PROGRAM Stn053_19_GrnRedRecircMergeSpurPrestop
VAR

	{attribute 'TcLinkToOSO' := '.iPuckPresent := <0,1,0>TIIB[N46S00 (AL1332)]^N46S03 (AL2341)^TxPDO^input byte 0;
								 .iBufferFull := <0,1,2>TIIB[N32S00 (AL1332)]^N32S05 (AL2341)^TxPDO^input byte 2;
								 .oStopLower := <0,1,4>TIIB[N46S00 (AL1332)]^N46S02 (EX260)^RxPDO^output byte 0'}
	fbConvStop: FB_ConvStop;
END_VAR

//MergeGrntoRedMergeSpurPrestopGrn  (3A)  VB10 Enc56 near Mtr 3 & 4 - bottom of High Friction Green conveyor
//GRNRED Recirc Merge GRN Stop Puck Present enc56 M1 H1  H3208
//EvalGRN RED Recirc Merge DS Buffer Full    H4423  Red Conv - Enc55  M2 H3

//  This code instantiates a component that is implimented as a common function block
//    Note that I/O is linked directly to I/O variables inside the named instance

gStn053_19_GrnRedRecircMergeSpurPrestop.ConvRunning  := gConsumed_SafetyInterfaceConv.MtrRunning.Enc056Mtr04;

fbConvStop(
	pStn := ADR(gStn053),
	pCmp := ADR(gStn053_19_GrnRedRecircMergeSpurPrestop),
	pUpstreamStop := 0,
	pStateTraceBuffer := ADR(gStn053_StateTraceBuffer),
	pStateTraceFifo := ADR(gStn053_StateTraceFifo),
	pStats := ADR(gStn053_02_Stats));

END_PROGRAM

(* stored: Version 1.1.0.1, ProductVersion 3.1.4024.6
   POU Stn053_19_GrnRedRecircMergeSpurPrestop: Id {b27251dc-e5eb-44b2-a7b5-8059706b9d47}, SpecialFunc None *)
